FUNCTION_BLOCK FB_influxdb
VAR_INPUT
	// Process is started at rising edge
	Trigger: BOOL;
	// table,e.g. thermocontrol
	table:	STRING;
	//e.g. dewar_pressure=1e-5, ...
	measurements: STRING;
	timeout: TIME := T#6S;
END_VAR
VAR_OUTPUT
	Busy:	BOOL;
	Error:	BOOL;
	ErrorID:	UDINT;
END_VAR
VAR
	curl: NT_StartProcess;
	arguments: STRING := '';
END_VAR
VAR CONSTANT
	prefix:	STRING(100) := '-i -XPOST "http://192.168.7.150:8086/write?db=bmkdb&precision=s" --connect-timeout 3 --data-binary ';
END_VAR

//curl -i -XPOST "http://192.168.7.206:8086/write?db=bmkdb&precision=s" --data-binary 'thermocontrol ...'
arguments := CONCAT('"', table);
arguments := CONCAT(arguments, ' ');
arguments := CONCAT(arguments, measurements);
arguments := CONCAT(arguments, '"');
curl(NETID	:=	'',
	PATHSTR	:=	'C:\bin\curl-7.65.3-win32-mingw\bin\curl.exe',
	DIRNAME	:=	'C:\bin\curl-7.65.3-win32-mingw\bin',
	COMNDLINE:=	CONCAT(prefix, arguments),
	START	:=	Trigger,
	TMOUT	:=	timeout,
	BUSY 	=>	Busy,
	ERR		=> Error,
	ERRID	=> ErrorID);

END_FUNCTION_BLOCK

(* stored: Version 1.1.0.1, ProductVersion 3.1.4024.0
   POU FB_influxdb: Id {1fea41b1-e692-4070-bc8f-e6709f9f4692}, SpecialFunc None *)
